GLOBALCONSTANTS AID_EXOP (* External object pointer object attribute ids *)
  (* Standard: 61499-1; Description: Copyright (c) 2023 HR Agrartechnik GmbH This program and the accompanying materials are made available under the terms of the Eclipse Public License 2.0 which is available at https://www.eclipse.org/legal/epl-2.0/ SPDX-License-Identifier: EPL-2.0 *)
  (* Version 1.0, 2026-06-20, Franz Höpfinger, HR Agrartechnik GmbH *)
  PACKAGE isobus::UT::Q::const::AID;
  VAR_GLOBAL CONSTANT
    DEF_OBJ_ID : USINT := USINT#1; (* 1: AID_EXOP_DEF_OBJ_ID - Default Object ID to display if external ID is not valid or is the NULL *)
    EXT_REF_NAME_ID : USINT := USINT#2; (* 2: AID_EXOP_EXT_REF_NAME_ID - Object id of an External Reference NAME object. *)
    EXT_OBJ : USINT := USINT#3; (* 3: AID_EXOP_EXT_OBJ *)
  END_VAR
END_GLOBALCONSTANTS
